# EPICS StreamDevice protocol: Chpt2/arduino.proto
Terminator = CR LF;

set_digital{
    out "%d";
    ExtraInput = Ignore;
}
